// Mitsubishi GX Works2 project: 시퀀스 예제 2_2   PLC: Q03UDV

PROGRAM MAIN
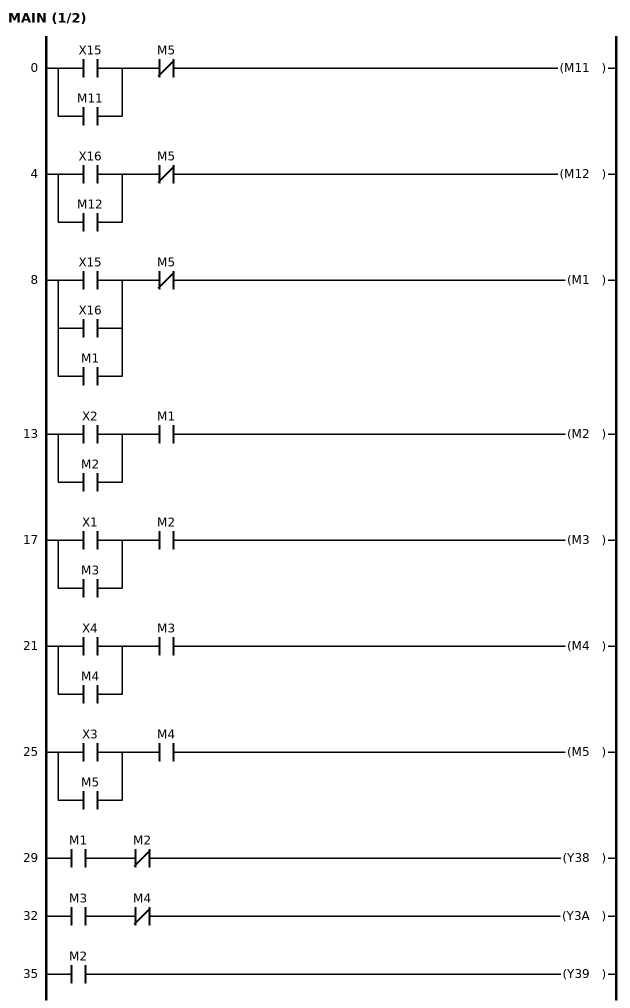
0     LD      X15
      OR      M11
      ANI     M5
      OUT     M11
4     LD      X16
      OR      M12
      ANI     M5
      OUT     M12
8     LD      X15
      OR      X16
      OR      M1
      ANI     M5
      OUT     M1
13    LD      X2
      OR      M2
      AND     M1
      OUT     M2
17    LD      X1
      OR      M3
      AND     M2
      OUT     M3
21    LD      X4
      OR      M4
      AND     M3
      OUT     M4
25    LD      X3
      OR      M5
      AND     M4
      OUT     M5
29    LD      M1
      ANI     M2
      OUT     Y38
32    LD      M3
      ANI     M4
      OUT     Y3A
35    LD      M2
      OUT     Y39
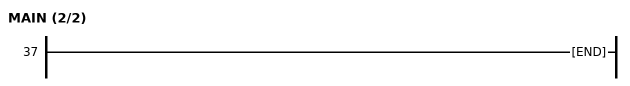
37    END
END_PROGRAM
